TYPE ST_BaseHMILoggerElement_Command :
STRUCT
END_STRUCT
END_TYPE

(* stored: Version 1.1.0.1
   DUT ST_BaseHMILoggerElement_Command: Id {f8918eb0-a077-0ca9-01f2-5f406b2b0692} *)
